{attribute 'qualified_only'}
VAR_GLOBAL
END_VAR

VAR_GLOBAL CONSTANT
	nAXIS_NUM			: 	UINT := 4;
END_VAR

(* stored: Version 1.1.0.1, ProductVersion 3.1.4024.5
   GVL GVL_APP: Id {8df35838-54af-476a-8669-93658e0ca478} *)
